// TIA Portal V16 export
// export: Created 2024-12-03T15:41:40.6259842Z, ExportSetting WithDefaults, DisplayName Totally Integrated Automation Portal, DisplayVersion V16 Update 6, DisplayName TIA Portal Version Control Interface, DisplayVersion V16 Update 2, DisplayName TIA Portal Openness, DisplayVersion V16 Update 6, DisplayName TIA Portal Teamcenter Gateway, DisplayVersion V16, DisplayName SINAMICS Startdrive Advanced, DisplayVersion V16 Update 5, DisplayName SINAMICS Startdrive G130, G150, S120, S150, SINAMICS MV, S210, DisplayVersion V16 Update 5, DisplayName SINAMICS Startdrive G110M, G120, G120C, G120D, G120P, G115D, DisplayVersion V16 Update 5, DisplayName STEP 7 Professional, DisplayVersion V16 Update 6, DisplayName STEP 7 Safety, DisplayVersion V16, DisplayName WinCC Advanced / Unified PC, DisplayVersion V16 Update 6
FUNCTION_BLOCK "InstallaitonControlInstance"   // FB67, SCL
{ S7_Optimized_Access := 'TRUE' }
VERSION : 0.1
// stored: AutoNumber true, IsIECCheckEnabled false, IsRetainMemResEnabled false, MemoryReserve 100, SetENOAutomatically false, UDAEnableTagReadback false
   VAR_IN_OUT
      IO_Appstate : "ApplicationState_UDT";
   END_VAR
   VAR
      HmiReset { S7_SetPoint := 'True'} : "HmiButton";
      HmiStartAutoMode { S7_SetPoint := 'True'} : "HmiButton";
      HmiStopAutoMode { S7_SetPoint := 'True'} : "HmiButton";
      HmiActivateManualMode { S7_SetPoint := 'True'} : "HmiButton";
      HmiDeactivateManualMode { S7_SetPoint := 'True'} : "HmiButton";
      HmiStartEmptyMode { S7_SetPoint := 'True'} : "HmiButton";
      HmiStopEmptyMode { S7_SetPoint := 'True'} : "HmiButton";
      HmiStandbyMode { S7_SetPoint := 'True'} : "HmiButton";
      AutModeActivated { S7_SetPoint := 'True'} : "SmartBool";
      ManualModeActivated { S7_SetPoint := 'True'} : "SmartBool";
      EmptyModeActivated { S7_SetPoint := 'True'} : "SmartBool";
      StandbyMode { S7_SetPoint := 'True'} : "SmartBool";
      OnDelayAutoMode { S7_SetPoint := 'True'} : TON_TIME;
   END_VAR
   VAR DB_SPECIFIC
      AutoMode : Bool;
      ManualMode : Bool;
      EmptyMode : Bool;
   END_VAR
   VAR
      Standby : Bool;
   END_VAR
   VAR_TEMP
      T_Index : Int;
      T_EnableButton : Bool;
      T_Appstate : "ApplicationState_UDT";
   END_VAR
BEGIN
   REGION HMI buttons

       REGION RESET

           IF "HMI_DB".ResetFromHMI THEN
               #IO_Appstate.Hmi_Buttons.reset.SignalFromHMI := 1;
           END_IF;

           #T_EnableButton := true;
           #HmiReset(I_Enable := #T_EnableButton,
                     ButtonStatus := #IO_Appstate.Hmi_Buttons.reset);

       END_REGION

       REGION RESET ALARM
           IF #IO_Appstate.Hmi_Buttons.reset.state.State THEN
               #IO_Appstate.Alarms.AlarmActiveInternalPLC := FALSE;
           END_IF;
       END_REGION

       REGION START AUTO MODE
           #T_EnableButton := (#IO_Appstate.States.ReadyForAutoMode
           OR  #IO_Appstate.States.ManaulOverrideActive.HMI)
           AND NOT #IO_Appstate.States.ManualModeActivated.State
           AND (NOT #IO_Appstate.States.AutoModeActivated.State OR #IO_Appstate.States.Standby.State);
           #T_EnableButton := #T_EnableButton AND #IO_Appstate.States.EmergencyOk.State;

           #HmiStartAutoMode(ButtonStatus := #IO_Appstate.Hmi_Buttons.StartAutoMode,
                             I_Enable := #T_EnableButton);
       END_REGION

       REGION STOP AUTO MODE
           #T_EnableButton := #IO_Appstate.States.AutoModeActivated.State;
           #T_EnableButton := #T_EnableButton AND #IO_Appstate.States.EmergencyOk.State;
           #HmiStopAutoMode(I_Enable := #T_EnableButton,
                            I_Flash := #IO_Appstate.States.RequestingAutoModeOff,
                            ButtonStatus := #IO_Appstate.Hmi_Buttons.StopAutoMode);
       END_REGION

       REGION standby mode
           #T_EnableButton := #IO_Appstate.States.AutoModeActivated.State;
           #T_EnableButton := #T_EnableButton AND #IO_Appstate.States.EmergencyOk.State;
           #HmiStandbyMode(I_Enable := #T_EnableButton,
                           ButtonStatus := #IO_Appstate.Hmi_Buttons.ActivateStandby);

       END_REGION

       REGION START MANUAL MODE
           #T_EnableButton := NOT #IO_Appstate.States.AutoModeActivated.State
           AND NOT #IO_Appstate.States.ManualModeActivated.State;
           #T_EnableButton := #T_EnableButton AND #IO_Appstate.States.EmergencyOk.State;
           #HmiActivateManualMode(I_Enable := #T_EnableButton,
                                  ButtonStatus := #IO_Appstate.Hmi_Buttons.ActivateManualMode);
       END_REGION

       REGION STOP MANUAL MODE
           #T_EnableButton := #IO_Appstate.States.ManualModeActivated.State;
           #T_EnableButton := #T_EnableButton AND #IO_Appstate.States.EmergencyOk.State;
           #HmiDeactivateManualMode(I_Enable := #T_EnableButton,
                                    ButtonStatus := #IO_Appstate.Hmi_Buttons.DeactivateManualMode);
       END_REGION

       REGION START EMPTY MODE
           #T_EnableButton := #IO_Appstate.States.AutoModeActivated.State AND NOT #IO_Appstate.States.EmptyApplicatoinMode.State;
           #T_EnableButton := #T_EnableButton AND #IO_Appstate.States.EmergencyOk.State;
           #HmiStartEmptyMode(I_Enable := #T_EnableButton,
                              ButtonStatus := #IO_Appstate.Hmi_Buttons.StartEmptyMode);
       END_REGION

       REGION STOP EMPRTY MODE
           #T_EnableButton := #IO_Appstate.States.EmptyApplicatoinMode.State;
           #T_EnableButton := #T_EnableButton AND #IO_Appstate.States.EmergencyOk.State;
           #HmiStopEmptyMode(I_Enable := #T_EnableButton,
                             ButtonStatus := #IO_Appstate.Hmi_Buttons.StopEmptyMode);
       END_REGION

   END_REGION

   REGION Auto mode

       #IO_Appstate.States.ReadyForAutoMode := true;

       IF #IO_Appstate.States.ManualModeActivated.State THEN
           #IO_Appstate.States.ReadyForAutoMode := false;
       END_IF;

       IF #IO_Appstate.Hmi_Buttons.StartAutoMode.state.LE AND #IO_Appstate.States.ReadyForAutoMode THEN
           #AutoMode := true;
       END_IF;

       IF #IO_Appstate.Hmi_Buttons.StopAutoMode.state.LE THEN
           #IO_Appstate.States.RequestingAutoModeOff := true;
       END_IF;

       IF (#IO_Appstate.States.RequestingAutoModeOff AND #IO_Appstate.States.ReadyForStandby)
           OR NOT #IO_Appstate.States.EmergencyOk.State THEN
           #AutoMode := FALSE;
       END_IF;

       IF NOT #AutoMode THEN
           #IO_Appstate.States.RequestingAutoModeOff := FALSE;
       END_IF;

       IF #IO_Appstate.States.ManualModeActivated.State THEN
          // OR NOT IO_Appstate.States.EmergencyOk.State THEN
           #AutoMode := false;
       END_IF;

       #OnDelayAutoMode(IN:=#AutoMode,
                        PT:=t#0s);

       #AutModeActivated(I_Sensor := #OnDelayAutoMode.Q,
                         O_data => #IO_Appstate.States.AutoModeActivated);

   END_REGION

   REGION STANDBY MODE

       IF #IO_Appstate.Hmi_Buttons.ActivateStandby.state.State AND #IO_Appstate.States.AutoModeActivated.State THEN
           #Standby := true;
       END_IF;

       IF #IO_Appstate.Hmi_Buttons.StartAutoMode.state.LE
           AND #IO_Appstate.States.Standby.State THEN
           #Standby := false;
       END_IF;

       IF NOT #AutoMode THEN
           #Standby := false;
       END_IF;

       #StandbyMode(I_Sensor := #Standby,
                    O_data => #IO_Appstate.States.Standby);

   END_REGION

   REGION Manual mode

       IF #IO_Appstate.Hmi_Buttons.ActivateManualMode.state.LE THEN
           #ManualMode := true;
       END_IF;

       IF #IO_Appstate."Hmi_Buttons".DeactivateManualMode.state.LE
           //OR NOT IO_Appstate.States.EmergencyOk.State
           OR #AutoMode THEN
           #ManualMode := FALSE;
       END_IF;

       #ManualModeActivated(I_Sensor := #ManualMode,
                            O_data => #IO_Appstate.States.ManualModeActivated);

   END_REGION

   REGION Empty Moode

       IF #IO_Appstate.Hmi_Buttons.StartEmptyMode.state.LE THEN
           #EmptyMode := true;
       END_IF;

       IF #IO_Appstate.Hmi_Buttons.StopEmptyMode.state.LE
           OR NOT #IO_Appstate.States.AutoModeActivated.State
           OR NOT #IO_Appstate.States.EmergencyOk.State THEN
           #EmptyMode := 0;
       END_IF;

       #EmptyModeActivated(I_Sensor := #EmptyMode,
                           O_data => #IO_Appstate.States.EmptyApplicatoinMode);

                            END_REGION

    REGION manaul override
        #IO_Appstate.States.ManaulOverrideActive.HMI := #IO_Appstate.States.ManaulOverrideActive.Internal;
        #IO_Appstate.States.ManaulOverrideActive.Internal := false;
    END_REGION

   REGION ALARMS

       #IO_Appstate.Alarms.AlarmsActiveForHmi := #IO_Appstate.Alarms.AlarmActiveInternalPLC;
       #IO_Appstate.Alarms.AlarmActiveInternalPLC := false;

   END_REGION
END_FUNCTION_BLOCK
